PROGRAM FunktionBlockDiagram
VAR
	
END_VAR

END_PROGRAM

(* stored: Version 1.1.0.1
   POU FunktionBlockDiagram: Id {bb9f87a0-c1f0-406b-9126-1016eb4ae4b7}, SpecialFunc None *)
